Staubli VAL3: setOnline.pgx

public program setOnline(num handle_, bool online_, bool& result_[])
begin
  // put camera into online or offline mode
  // online_ : if true put camera online
  //           if false put camera to offline
  // result_ : result of operation
  nCommand[handle_]=coSO
  if online_
    call sendCommand(handle_,"so1",result_)
  else
    call sendCommand(handle_,"so0",result_)
  endIf
end
